Staubli VAL3: onStop.pgx

public program onStop(string& x_sItem[])
begin
  // stop it
  if x_sItem=="kill"
    pt:libLoad("Disk://kernel/template/session/saveTraj/POINT")
  endIf
end
